FUNCTION_BLOCK UA_MethodCall_ADSReadStateReq
VAR_INPUT
	bExecute			: BOOL;
	nConnectionHdl		: DWORD;
	nNamespaceIndex		: UINT; 			(* to be retrieved using UA_GetNamespaceIndex *)
	sNetID				: T_AmsNetId; 		(* AmsNetId OF the Target *)
	nPort				: INT; 			(* Port number	*)
	cbData				: UDINT;			(* Count OF bytes to be read*)
	pData				: PVOID;
	Timeout				: TIME := DEFAULT_ADS_TIMEOUT;
END_VAR
VAR_OUTPUT
	nAdsState			: DINT;			(* ADS state *)
	nDeviceState		: DINT;			(* Device state *)
	cbReadData_R		: UDINT; 
	bDone				: BOOL;
	bBusy				: BOOL;
	bError				: BOOL;
	nErrorID			: DWORD;
END_VAR
VAR
	iReadStateReqState	: INT;
	RTrig				: R_TRIG;

	fbUA_MethodGetHandle: UA_MethodGetHandle;
	nMethodHdl			: DWORD;
	ObjectNodeID		: ST_UANodeID;
	MethodNodeID		: ST_UANodeID;

	fbUA_MethodCall		: UA_MethodCall;
	InputArguments		: ARRAY [1..nNumberOfInputArguments] OF ST_UAMethodArgInfo; (*ReadStateReq has 2 input parameters *)
	stOutputArgInfoAndData	: ST_UAMethodCall_AdsReadStateRes; // (4+OutputArgInfo+8)bytes
	stOutputArgInfo		: ARRAY [1..nNumberOfOutputArguments] OF ST_UAMethodArgInfo;
	
	nArg				: INT;
	nInputData			: ARRAY [1..nInputArgSize] OF BYTE; (* NetID(24) + Port(2) *)
	nOffset				: UDINT;
	
	fbUA_MethodReleaseHandle	: UA_MethodReleaseHandle;
	bInputDataError 			: BOOL;
END_VAR
VAR CONSTANT
	nInputArgSize				: UDINT := 26; (* NetID(24) + Port(2) *)
	nNumberOfInputArguments 	: UDINT := 2;
	nNumberOfOutputArguments	: UDINT := 3;
END_VAR

(*
ADSReadStateReq(
******** Input Arguments ********
	string sNetID, 		: AmsNetId of the Target
	int16 Port,			: Port number	
	
******** Output Arguments ********
	int32 AdsState,		: Ads State
	int32 DeviceState	: Device State
	ByteString Data		: Data
);
*)


RTrig(CLK:= bExecute);

CASE iReadStateReqState OF

0:	(* Get Method Handle *)
	IF RTrig.Q THEN
		bBusy	:= TRUE;
		bDone 	:= FALSE;
		bError	:= FALSE;
		nErrorID	:= 0;
		ObjectNodeID.eIdentifierType 	:= eUAIdentifierType_String;
		ObjectNodeID.nNamespaceIndex 	:= nNamespaceIndex;
		ObjectNodeID.sIdentifier		:= 'ADSAMS';
	
		MethodNodeID.eIdentifierType 	:= eUAIdentifierType_String;
		MethodNodeID.nNamespaceIndex 	:= nNamespaceIndex;
		MethodNodeID.sIdentifier		:= 'ADSAMS.AdsReadStateReq';
		
		M_Init();
		IF bInputDataError = FALSE THEN
			iReadStateReqState 	:= iReadStateReqState + 1;
		ELSE
			bBusy 		:= FALSE; 
			bError 		:= TRUE;
			nErrorID 	:= DEVICE_INVALIDSIZE; //16#705 parameter size not correct
		END_IF
		nAdsState		:= 0;			(* ADS state *)
		nDeviceState	:= 0;			(* Device state *)
	END_IF


1:	(* Method Get Handle *)
	fbUA_MethodGetHandle(
			Execute			:= TRUE,
			ConnectionHdl	:= nConnectionHdl,
			ObjectNodeID	:= ObjectNodeID,
			MethodNodeID 	:= MethodNodeID,
			Timeout			:= Timeout,
			MethodHdl		=> nMethodHdl
		);
	IF NOT fbUA_MethodGetHandle.Busy THEN
		fbUA_MethodGetHandle(Execute := FALSE);

		IF NOT fbUA_MethodGetHandle.Error THEN
			(*  *)
			iReadStateReqState 	:= iReadStateReqState + 1; (* Call Method *)
		ELSE
			bError				:= TRUE;
			nErrorID			:= fbUA_MethodGetHandle.ErrorID;
			iReadStateReqState 	:= 3; (* Release Handle *)
		END_IF
	END_IF


2:	(* Method Call *)
	fbUA_MethodCall(
		Execute					:= TRUE,
		ConnectionHdl			:= nConnectionHdl,
		MethodHdl				:= nMethodHdl,
		nNumberOfInputArguments := nNumberOfInputArguments,		(* 2 *)
		pInputArgInfo			:= ADR(InputArguments),
		cbInputArgInfo			:= SIZEOF(InputArguments),
		pInputArgData			:= ADR(nInputData),
		cbInputArgData			:= nOffset,
		pInputWriteData			:= 0,
		cbInputWriteData		:= 0,
		nNumberOfOutputArguments:= nNumberOfOutputArguments,	(* 3 *)
		pOutputArgInfo			:= ADR(stOutputArgInfo),
		cbOutputArgInfo			:= SIZEOF(stOutputArgInfo),
		pOutputArgInfoAndData	:= ADR(stOutputArgInfoAndData),
		cbOutputArgInfoAndData	:= SIZEOF(stOutputArgInfoAndData),
		Timeout					:= Timeout
	);
	IF NOT fbUA_MethodCall.Busy THEN
		fbUA_MethodCall(Execute := FALSE, cbRead_R => cbReadData_R);

		IF NOT fbUA_MethodCall.Error THEN
			(*  *)
			iReadStateReqState 	:= iReadStateReqState + 1; (* Release handle *)
			nAdsState := stOutputArgInfoAndData.stADSReadState.nAdsState;
			nDeviceState := stOutputArgInfoAndData.stADSReadState.nDeviceState;		
		ELSE
			bError				:= TRUE;
			nErrorID			:= fbUA_MethodCall.ErrorID;
			iReadStateReqState 	:= 3; (* Release handle *)
		END_IF
	END_IF


3:	(* Release Method Handle *)
	fbUA_MethodReleaseHandle(
		Execute			:= TRUE,
		ConnectionHdl	:= nConnectionHdl,
		MethodHdl		:= nMethodHdl,
		Timeout			:= Timeout
	);

	IF NOT fbUA_MethodReleaseHandle.Busy THEN
		fbUA_MethodReleaseHandle(Execute := FALSE);
		bBusy := FALSE;
		IF NOT fbUA_MethodReleaseHandle.Error THEN
			(* session closed *)
			bDone := TRUE;
			iReadStateReqState 	:= 0; (* idle *)
		ELSE
			bError				:= TRUE;
			nErrorID			:= fbUA_MethodReleaseHandle.ErrorID;
			iReadStateReqState 	:= 0; (* idle *)
		END_IF
	END_IF
END_CASE

ACTION M_Init:
bInputDataError := FALSE; 
nOffset := 0;
MEMSET(ADR(InputArguments),0,SIZEOF(InputArguments));
MEMSET(ADR(nInputData),0,SIZEOF(nInputData));

nArg := 1;
(*sNetID := sAmsNetID;*)	(********** NET ID **********)
InputArguments[nArg].DataType			:= eUAType_String;
InputArguments[nArg].ValueRank			:= -1; 						(* Scalar = -1 or Array *)
InputArguments[nArg].ArrayDimensions[1]	:= 0; 						(* Number of Dimension in case its an array *)
InputArguments[nArg].nLenData			:= INT_TO_UDINT(LEN(sNetId)) + 1;			(* Length if its a STRING *)
IF nOffset + INT_TO_UDINT(LEN(sNetId))+1 > nInputArgSize THEN 
	bInputDataError := TRUE;
	RETURN;
ELSE
	MEMCPY(ADR(nInputData)+nOffset,ADR(sNetId),INT_TO_UDINT(LEN(sNetId))+1);				(* VALUE in BYTES FORM *)
	nOffset := nOffset + INT_TO_UDINT(LEN(sNetId))+1;
END_IF

nArg := nArg + 1;
(* nPort := 851;*)			(********** PORT **********)
InputArguments[nArg].DataType			:= eUAType_Int16;
InputArguments[nArg].ValueRank			:= -1; 						(* Scalar = -1 or Array *)
InputArguments[nArg].ArrayDimensions[1]	:= 0; 						(* Number of Dimension in case its an array *)
InputArguments[nArg].nLenData			:= SIZEOF(nPort);			(* Length if its a STRING *)
IF nOffset + SIZEOF(nPort) > nInputArgSize THEN 
	bInputDataError := TRUE;
	RETURN;
ELSE
	MEMCPY(ADR(nInputData)+nOffset,ADR(nPort),SIZEOF(nPort));			(* VALUE in BYTES FORM *)
	nOffset := nOffset + SIZEOF(nPort);
END_IF

//************** Prepare Output Argument information ***********
stOutputArgInfo[1].nLenData := SIZEOF(stOutputArgInfoAndData.stADSReadState.nAdsState);
stOutputArgInfo[2].nLenData := SIZEOF(stOutputArgInfoAndData.stADSReadState.nDeviceState); 
stOutputArgInfo[3].nLenData := 0;
END_ACTION

END_FUNCTION_BLOCK

(* stored: Version 1.1.0.1, ProductVersion 3.1.4022.6
   POU UA_MethodCall_ADSReadStateReq: Id {f0dd222a-7fd2-4963-8e28-5f9668204f23}, SpecialFunc None
   Action M_Init: Id {fc735a50-8d23-449b-8c67-528c6d874c24} *)
